FUNCTION_BLOCK FB_ComponentBase IMPLEMENTS ITF_ComponentBase
VAR_INPUT
END_VAR
VAR_OUTPUT
END_VAR
VAR CONSTANT
	//Constant declarations
	COMPONENT_BASE_ALARM_COUNT	: UDINT := 16;
END_VAR

VAR	
	//ITF_BasicComponent internal property variables
	bError 			: BOOL;			//Boolean to signal that an error has ocurred
	nErrorID 		: UDINT;		//Integer ID to identify the proper alarm to be posted from the parent module
	bEnabled		: BOOL;			//Enables or disables the component
	bSimulate		: BOOL;			//TRUE disables all hardware I/O and simulates input and output behavior
	sName			: STRING;		//String name of the component
	bActive			: BOOL;			//TRUE when the component is in its energized state, motion or detection
	
	//Alarming
	a_fbComponentBaseAlarms : ARRAY[1..COMPONENT_BASE_ALARM_COUNT] OF FB_TcAlarm;
	
	//HMI Monitoring and control structure
	stComponentBaseHMI : ST_ComponentBase_HMI;
	
	//Internal Variables
	bInitialized	: BOOL;
	
END_VAR

PROPERTY Active : BOOL	//TRUE when the component is in motion or otherwise completing a commanded task
GET
Active := bActive;
END_GET
END_PROPERTY

METHOD CyclicLogic : BOOL		//Should be called Externally akin to the PML Modules
IF NOT bInitialized THEN
	initialize();
	bInitialized := TRUE;
END_IF

IF NOT bSimulate AND NOT bError THEN	//If not in simulation mode or error state
	StandardOperation();
ELSIF NOT bError THEN
	SimulateOperation();	//Simulate inputs and outputs
ELSE
	ErrorOperation();
END_IF

Monitoring();		//Constant error and status monitoring
HardwareUpdate();	//Passes internal commands to hardware outputs and vice versa for inputs, implement via extended FB override
HMICommunication();	//Keeps the HMI data up to date, and processes requests from the HMI for this component
END_METHOD

PROPERTY Enabled : BOOL	//Enables or disables the component
GET
Enabled := bEnabled;
END_GET
SET
bEnabled := Enabled;
END_SET
END_PROPERTY

PROPERTY Error : BOOL	//Boolean to signal that an error has ocurred
GET
Error := bError;
END_GET
END_PROPERTY

PROPERTY ErrorID : UDINT	//Integer ID to identify the proper alarm to be posted from the parent module
GET
ErrorID := nErrorID;
END_GET
SET
nErrorID := ErrorID;
END_SET
END_PROPERTY

METHOD ErrorOperation : BOOL
VAR_INPUT
END_VAR
//Override from extended FB with error operation logic (Shut off outputs, clear inputs, blink, send error messages, etc)
END_METHOD

METHOD HardwareUpdate : BOOL
VAR_INPUT
END_VAR
//override from extended FB with reads and writes between internal variables and hardware inputs and outputs
END_METHOD

METHOD HMICommunication : BOOL
//Extend this method in extended FBs to communicate specific implementation data

//Process HMI requests
IF stComponentBaseHMI.bIncomingHMIRequest AND NOT stComponentBaseHMI.bHMICommandConfirmation THEN		//If a request has been issued by the HMI, and a previous request has not just finished being processed
	IF stComponentBaseHMI.bHMIControlAvailable THEN		//If the current conditions permit HMI control (Should be determined by the extended application components)
		IF stComponentBaseHMI.bEnableHMIRequest THEN
			bEnabled := TRUE;
			stComponentBaseHMI.bHMICommandConfirmation := TRUE;	//Confirm that the request has been processed
		END_IF
		IF stComponentBaseHMI.bDisableHMIRequest THEN
			bEnabled := FALSE;
			stComponentBaseHMI.bHMICommandConfirmation := TRUE;	//Confirm that the request has been processed
		END_IF
		IF stComponentBaseHMI.bResetHMIRequest THEN
			Reset();
			stComponentBaseHMI.bHMICommandConfirmation := TRUE;	//Confirm that the request has been processed
		END_IF
		IF stComponentBaseHMI.bSimulateOperationHMIRequest THEN
			bSimulate := TRUE;
			stComponentBaseHMI.bHMICommandConfirmation := TRUE;	//Confirm that the request has been processed
		END_IF
		IF stComponentBaseHMI.bStandardOperationHMIRequest THEN
			bSimulate := FALSE;
			stComponentBaseHMI.bHMICommandConfirmation := TRUE;	//Confirm that the request has been processed
		END_IF
	END_IF
END_IF

//Update HMI status info
stComponentBaseHMI.bActive := bActive;
stComponentBaseHMI.bEnabled := bEnabled;
stComponentBaseHMI.sName := sName;
stComponentBaseHMI.bError := bError;
stComponentBaseHMI.bSimulate := bSimulate;
stComponentBaseHMI.nErrorID := nErrorID;
END_METHOD

METHOD initialize : BOOL
VAR_INPUT
END_VAR

VAR
	sTemp: STRING;
END_VAR
//Extend initialize as needed in extended FBs

sTemp := CONCAT(CONCAT(CONCAT('Component ', ': '), sName), ' '); 	//Creates a utility string for alarms and other messaging that reads (example text) - "Module 10 - Main Casepacker" to be followed by the alarm or message info
//TODO: Rename Event Class to AxisBase
F_CreateAllEventsInClass(	p_aAlarms := a_fbComponentBaseAlarms,
							nClassSize := SIZEOF(TC_EVENTS.ComponentBase),
							pInitEvent := ADR(TC_EVENTS.ComponentBase.InitReferenceEvent),
							sPrefix := sTemp );
END_METHOD

METHOD Monitoring : BOOL
VAR_INPUT
END_VAR
//Override/extend from extended FB with monitoring logic
END_METHOD

PROPERTY Name : STRING
GET
Name := sName;
END_GET
SET
sName := Name;
END_SET
END_PROPERTY

METHOD Reset : BOOL
bError := FALSE;
nErrorID := 0;
END_METHOD

{warning 'add property implementation'}
PROPERTY Simulate : BOOL
GET
Simulate := bSimulate;
END_GET
SET
bSimulate := Simulate;
END_SET
END_PROPERTY

METHOD SimulateOperation : BOOL
VAR_INPUT
END_VAR
//Override from extended FB with simulated operation logic
IF bEnabled THEN
	//Do Stuff
	;
ELSE
	//Don't Do Stuff
	;
END_IF
END_METHOD

METHOD StandardOperation : BOOL
VAR_INPUT
END_VAR
//Override from extended FB with normal operation logic
IF bEnabled THEN
	//Do Stuff
	;
ELSE
	//Don't Do Stuff
	;
END_IF
END_METHOD

END_FUNCTION_BLOCK

(* stored: Version 1.1.0.1, ProductVersion 3.1.4024.9
   POU FB_ComponentBase: Id {93c9c074-e59b-49de-8b78-d1cf33f60885}, SpecialFunc None
   Folder 01_ITF_ComponentBase: Id {c6d497f2-156e-440d-9c2c-1c03eea21d72}
   Folder 01_Properties: Id {e5c64086-407c-425b-a16b-0d3b6dfdd425}
   Folder 01_Config: Id {7f5fe1c6-7354-4325-bb6d-2930dc36c8af}
   Folder 02_Control: Id {976c348b-cc04-4ee2-b1c7-700723149e3a}
   Folder 03_Status: Id {662f6474-0b26-4eab-937f-58c3c9eff2fd}
   Folder 02_Methods: Id {256a27d0-cb20-46ab-abcb-85152c0ab3db}
   Property Active: Id {bc61300b-bb09-450c-b21b-4eade2439fcc}
   Get Get: Id {22c6670c-3757-4ee9-9a04-bdbc7a7dc310}
   Method CyclicLogic: Id {afd9b957-a135-4679-8622-fc5b52009de2}
   Property Enabled: Id {86698bf0-894b-412a-87e8-32a70ab8aadb}
   Get Get: Id {1584ecb4-0ab9-4ebc-92c7-f70141f516a0}
   Set Set: Id {0418f117-1ae9-4e07-b1bf-c5eef8bb8881}
   Property Error: Id {6c90baf7-eb06-4116-9da9-d962bbb4001b}
   Get Get: Id {8302f893-6dd6-4501-9f37-3be08d29cf06}
   Property ErrorID: Id {522f54a0-4f42-4f97-93a1-3d636ade75ec}
   Get Get: Id {31491cde-d744-4c54-b94d-ebc7c59d30ac}
   Set Set: Id {520dc520-ad3e-4d52-a8b4-1551a2a50971}
   Method ErrorOperation: Id {f619ffd8-c4fa-4b59-8760-8523dde09884}
   Method HardwareUpdate: Id {abdd4852-be45-40a6-988f-bbe025414073}
   Method HMICommunication: Id {1d2523ef-921c-4ac8-8add-7cf4a36da1ba}
   Method initialize: Id {1cd968e9-db2d-41e3-8a70-d048b41b074e}
   Method Monitoring: Id {bfd9d149-0427-4d13-a652-4580ad3b7638}
   Property Name: Id {8d65d0ee-79e5-44fd-9af0-abf9b261fcfa}
   Get Get: Id {730ced66-cd8b-4cdd-b343-9360b6ba9ca2}
   Set Set: Id {265a41da-87cb-4c50-a4fb-f10a6353512e}
   Method Reset: Id {fdbb4a8b-7401-4011-85e0-df5c0eb6b89d}
   Property Simulate: Id {ebb42854-1266-4f6c-84a1-4c0a912b758b}
   Get Get: Id {17d1377a-ffdb-4d07-8b8e-165928f3cf8f}
   Set Set: Id {8823fd28-0770-436d-aba3-dbafa54451f7}
   Method SimulateOperation: Id {3671ca9e-3bc3-423d-9ff5-9067bbee6b2e}
   Method StandardOperation: Id {39013a93-6488-4d2f-b227-6a329265cedd} *)
